// TIA Portal V20 export
DATA_BLOCK "Config"   // DB195
// stored: MemoryReserve 100, Namespace Unit1
   VAR
      unit : "LAF_typeUnitConfiguration";   // Configuration of Unit Parameters
      stateMachine : "LUC_typeStateMachineConfiguration";
      signalStack : "LUC_typeSignalStackConfiguration";
      remoteCtrlOpcUa : "LUC_typeRemoteCtrlConfiguration";
      stateModeManager { ExternalAccessible := 'False'; ExternalVisible := 'False'; ExternalWritable := 'False'} : "LPMLV2022_typeConfiguration";   // Do not change. Can be configured through stateMachineConfiguration
      SLM : HW_SUBMODULE;
      cmFFU : "LER_typeLIU117Configuration";
      "========Communication========" : Bool;
      BA030 : "LER_typeCommunicationConfiguration";
      BA040 : "LER_typeCommunicationConfiguration";
   END_VAR
BEGIN
   unit.referenceDesignator.relative := WSTRING#'U1';
   stateMachine.enableModes.noMode := true;
   stateMachine.enableModes.sleep := true;
   stateMachine.enableModes.deepSleep := true;
   stateMachine.enableModes.userMode04 := false;
END_DATA_BLOCK
